TYPE csp_caser_feed_magazine_ls_belt_status_enum :(
	CSP_CASE_FEED_MAGAZINE_LS_BELT_STATUS_NOT_INITIALIZED 							:= 0,
	CSP_CASE_FEED_MAGAZINE_LS_BELT_STATUS_DISABLED 									:= 10,
	CSP_CASE_FEED_MAGAZINE_LS_BELT_STATUS_ENABLE_REQUEST 							:= 70,
	CSP_CASE_FEED_MAGAZINE_LS_BELT_STATUS_ENABLING 									:= 80,
	CSP_CASE_FEED_MAGAZINE_LS_BELT_STATUS_ENABLED 									:= 100,
	CSP_CASE_FEED_MAGAZINE_LS_BELT_STATUS_RUNNING									:= 110,
	CSP_CASE_FEED_MAGAZINE_LS_BELT_STATUS_STOP_REQUEST 								:= 500,
	CSP_CASE_FEED_MAGAZINE_LS_BELT_STATUS_DISABLE_REQUEST 							:= 530,
	CSP_CASE_FEED_MAGAZINE_LS_BELT_STATUS_DISABLING 								:= 540
	) := CSP_CASE_FEED_MAGAZINE_LS_BELT_STATUS_NOT_INITIALIZED;
END_TYPE

(* stored: Version 1.1.0.1, ProductVersion 3.1.4024.3
   DUT csp_caser_feed_magazine_ls_belt_status_enum: Id {711981bb-7901-4392-b047-bc69142b74c6} *)
